Staubli VAL3: cycle_isLock.pgx

program cycle_isLock(bool& x_bLock[] (dimensions=1))
begin
  //
  // ask for the PLC lock status
  //
  x_bLock=cycleStatus:bPausePLC
end
